Staubli VAL3: INT_EDIT.pgx

program Int_Edit(num& x_nData, num x_nX, num x_nY)
  local num l_nKey
  local num l_nNum
begin

  call Int_EditS(x_nData,x_nX,x_nY,"")
end
